TYPE ST_Axis :
STRUCT
	
OUTPUT	:	ST_AxisOUT;
INPUT	:	ST_AxisIN;

END_STRUCT
END_TYPE

(* stored: Version 1.1.0.1, ProductVersion 3.1.4022.18
   DUT ST_Axis: Id {4a856dc4-a0d6-428b-a658-8c80bfa9950a} *)
